(* IEC 61131-3 sources: verifaps-lib/share/xPPU (part 14) *)

        STEP White : (*Local Id: 11 *)
            Set_PriorityWhite(N);
        END_STEP

        STEP Conveyor : (*Local Id: 15 *)
        END_STEP

        STEP Black : (*Local Id: 26 *)
            Set_PriorityBlack(N);
        END_STEP

        STEP Ramp_End : (*Local Id: 30 *)
        END_STEP

        STEP Metallic : (*Local Id: 43 *)
            Set_PriorityMetallic(N);
        END_STEP

        STEP SetTargetChanged : (*Local Id: 53 *)
        END_STEP
        TRANSITION FROM (ResetTargets) TO (White) := (WPType_White); END_TRANSITION
        TRANSITION FROM (ResetTargets) TO (Black) := (WPType_Black); END_TRANSITION
        TRANSITION FROM (ResetTargets) TO (Metallic) := (WPType_Metallic); END_TRANSITION
        TRANSITION FROM (ResetTargets) TO (White) := (WPType_White); END_TRANSITION
        TRANSITION FROM (ResetTargets) TO (Black) := (WPType_Black); END_TRANSITION
        TRANSITION FROM (White) TO (Conveyor) := (Priority_White=1); END_TRANSITION
        TRANSITION FROM (White) TO (Ramp_End) := (Priority_White=2); END_TRANSITION
        TRANSITION FROM (Black) TO (Ramp_End) := (Priority_Black=2); END_TRANSITION
        TRANSITION FROM (Black) TO (Conveyor) := (Priority_Black=1); END_TRANSITION
        TRANSITION FROM (Metallic) TO (Conveyor) := (Priority_Metallic=1); END_TRANSITION
        TRANSITION FROM (Metallic) TO (Ramp_End) := (Priority_Metallic=2); END_TRANSITION
        TRANSITION FROM (Conveyor) TO (SetTargetChanged) := (CurrentTarget_Conveyor); END_TRANSITION
        TRANSITION FROM (Ramp_End) TO (SetTargetChanged) := (CurrentTarget_Conveyor); END_TRANSITION
        TRANSITION FROM (Ramp_End) TO (SetTargetChanged) := (CurrentTarget_Ramp); END_TRANSITION
        TRANSITION FROM (Conveyor) TO (SetTargetChanged) := (CurrentTarget_Ramp); END_TRANSITION
        TRANSITION FROM (Conveyor) TO (SetTargetChanged) := (CurrentTarget_Conveyor); END_TRANSITION
        TRANSITION FROM (Ramp_End) TO (SetTargetChanged) := (CurrentTarget_Conveyor); END_TRANSITION
        TRANSITION FROM (Conveyor) TO (SetTargetChanged) := (CurrentTarget_Conveyor); END_TRANSITION
        TRANSITION FROM (Ramp_End) TO (SetTargetChanged) := (CurrentTarget_Conveyor); END_TRANSITION
        TRANSITION FROM (ACT_ChangeTarget_Init) TO (ResetTargets) := (NOT TargetChanged AND NOT GVL.IsSFCResetting); END_TRANSITION
        TRANSITION FROM (SetTargetChanged) TO (ACT_ChangeTarget_Init) := (TargetChanged); END_TRANSITION
    END_ACTION
    ACTION ACT_CheckWPType

        INITIAL_STEP Conveyor_ACT_CheckWPType_Init : (*Local Id: 0 *)
        END_STEP

        STEP Reset_WPType : (*Local Id: 3 *)
        END_STEP

        STEP Wait_a_little_bit : (*Local Id: 11 *)
        END_STEP

        STEP WP_Is_White : (*Local Id: 15 *)
        END_STEP

        STEP WP_Is_Metallic : (*Local Id: 22 *)
        END_STEP

        STEP WP_Is_Black : (*Local Id: 30 *)
        END_STEP

        STEP WP_Type_Checked : (*Local Id: 36 *)
        END_STEP
        TRANSITION FROM (Reset_WPType) TO (Wait_a_little_bit) := (OptSensor.DI_WPLight); END_TRANSITION
        TRANSITION FROM (Reset_WPType) TO (WP_Is_Black) := (Reset_WPType.t>T#1s AND NOT IndSensor.DI_WPMetallic AND NOT OptSensor.DI_WPLight); END_TRANSITION
        TRANSITION FROM (Wait_a_little_bit) TO (WP_Is_White) := (Wait_a_little_bit.t>T#100ms AND NOT IndSensor.DI_WPMetallic); END_TRANSITION
        TRANSITION FROM (Wait_a_little_bit) TO (WP_Is_Metallic) := (IndSensor.DI_WPMetallic); END_TRANSITION
        TRANSITION FROM (WP_Is_White) TO (WP_Type_Checked) := (WPType_White); END_TRANSITION
        TRANSITION FROM (WP_Is_Metallic) TO (WP_Type_Checked) := (WPType_Metallic); END_TRANSITION
        TRANSITION FROM (WP_Is_White) TO (WP_Type_Checked) := (WPType_White); END_TRANSITION
        TRANSITION FROM (WP_Is_Metallic) TO (WP_Type_Checked) := (WPType_Metallic); END_TRANSITION
        TRANSITION FROM (WP_Is_Black) TO (WP_Type_Checked) := (WPType_Black); END_TRANSITION
        TRANSITION FROM (Conveyor_ACT_CheckWPType_Init) TO (Reset_WPType) := (NOT WPTypeChecked AND NOT GVL.IsSFCResetting); END_TRANSITION
        TRANSITION FROM (WP_Type_Checked) TO (Conveyor_ACT_CheckWPType_Init) := (WPTypeChecked); END_TRANSITION
    END_ACTION
    ACTION ACT_SortWP

        INITIAL_STEP Init_ACT_SortWP : (*Local Id: 0 *)
        END_STEP

        STEP ConveyorForwards : (*Local Id: 3 *)
            Motor.ACT_TurnClockwise(N);
        END_STEP

        STEP Wait : (*Local Id: 6 *)
        END_STEP

        STEP Checking_WP_Type : (*Local Id: 9 *)
            ACT_CheckWPType(N);
        END_STEP

        STEP Changing_Target : (*Local Id: 12 *)
            ACT_ChangeTarget(N);
        END_STEP

        STEP Chose_Right_Destination : (*Local Id: 15 *)
        END_STEP

        STEP Switch_Extending : (*Local Id: 19 *)
            Switch.ACT_Extend(N);
        END_STEP

        STEP Allow_FollowConveyorToOperate : (*Local Id: 22 *)
        END_STEP

        STEP Wait2sec : (*Local Id: 27 *)
        END_STEP

        STEP Stop_Allowence : (*Local Id: 30 *)
        END_STEP

        STEP Switch_Retracting : (*Local Id: 35 *)
            Switch.ACT_Retract(N);
        END_STEP

        STEP Transporting_To_Ramp : (*Local Id: 40 *)
        END_STEP

        STEP TurnConveyorOff : (*Local Id: 44 *)
            Motor.ACT_Stop(N);
        END_STEP

        STEP WP_Is_Sorted : (*Local Id: 47 *)
        END_STEP
        TRANSITION FROM (Chose_Right_Destination) TO (Switch_Extending) := (CurrentTarget_Conveyor); END_TRANSITION
        TRANSITION FROM (Chose_Right_Destination) TO (Transporting_To_Ramp) := (CurrentTarget_Ramp); END_TRANSITION
        TRANSITION FROM (Switch_Retracting) TO (TurnConveyorOff) := (Switch.Retracted); END_TRANSITION
        TRANSITION FROM (Transporting_To_Ramp) TO (TurnConveyorOff) := (Transporting_To_Ramp.t>T#2s); END_TRANSITION
        TRANSITION FROM (Init_ACT_SortWP) TO (ConveyorForwards) := (NOT WPSorted AND NOT GVL.IsSFCResetting); END_TRANSITION
        TRANSITION FROM (ConveyorForwards) TO (Wait) := (Motor.TurningClockwise); END_TRANSITION
        TRANSITION FROM (Wait) TO (Checking_WP_Type) := (Wait.t>T#900ms OR IndSensor.DI_WPMetallic OR OptSensor.DI_WPLight); END_TRANSITION
        TRANSITION FROM (Checking_WP_Type) TO (Changing_Target) := (WPTypeChecked); END_TRANSITION
        TRANSITION FROM (Changing_Target) TO (Chose_Right_Destination) := (TargetChanged); END_TRANSITION
        TRANSITION FROM (Switch_Extending) TO (Allow_FollowConveyorToOperate) := (Switch.Extended); END_TRANSITION
        TRANSITION FROM (Allow_FollowConveyorToOperate) TO (Wait2sec) := (FollowConveyor_AllowedToOperate); END_TRANSITION
        TRANSITION FROM (Wait2sec) TO (Stop_Allowence) := (Wait2sec.t>T#2s); END_TRANSITION
        TRANSITION FROM (Stop_Allowence) TO (Switch_Retracting) := (NOT FollowConveyor_AllowedToOperate); END_TRANSITION
        TRANSITION FROM (TurnConveyorOff) TO (WP_Is_Sorted) := (Motor.Stopped); END_TRANSITION
        TRANSITION FROM (WP_Is_Sorted) TO (Init_ACT_SortWP) := (WPSorted); END_TRANSITION
    END_ACTION
    ACTION ACT_AutomaticExecute

        INITIAL_STEP SmallSortingConveyor_ACT_AutomaticExecute_Init : (*Local Id: 0 *)
        END_STEP

        STEP Interstep : (*Local Id: 3 *)
        END_STEP

        STEP Sort_WP : (*Local Id: 11 *)
            ACT_SortWP(N);
        END_STEP

        STEP SetAutomaticExecuteCompleted : (*Local Id: 14 *)
        END_STEP
        TRANSITION FROM (Interstep) TO (Sort_WP) := (Check_AllowedToOperate AND Interstep.t>T#500ms); END_TRANSITION
        TRANSITION FROM (Interstep) TO (SmallSortingConveyor_ACT_AutomaticExecute_Init) := (NOT Check_AllowedToOperate AND Interstep.t>T#500ms); END_TRANSITION
        TRANSITION FROM (Interstep) TO (Sort_WP) := (Check_AllowedToOperate AND Interstep.t>T#500ms); END_TRANSITION
        TRANSITION FROM (SmallSortingConveyor_ACT_AutomaticExecute_Init) TO (Interstep) := (Check_AllowedToOperate AND NOT AutomaticExecuteCompleted AND NOT GVL.IsSFCResetting); END_TRANSITION
        TRANSITION FROM (Sort_WP) TO (SetAutomaticExecuteCompleted) := (WPSorted); END_TRANSITION
        TRANSITION FROM (SetAutomaticExecuteCompleted) TO (SmallSortingConveyor_ACT_AutomaticExecute_Init) := (AutomaticExecuteCompleted); END_TRANSITION
    END_ACTION
    ACTION ACT_EmergencyStop

        INITIAL_STEP Conveyor_ACT_EmergencyStop_Init : (*Local Id: 0 *)
        END_STEP

        STEP ResetVariables : (*Local Id: 3 *)
            Reset_Variables(N);
        END_STEP

        STEP Stop_Conveyor : (*Local Id: 6 *)
            Motor.ACT_Stop(N);
        END_STEP

        STEP Retract_Switch : (*Local Id: 9 *)
            Switch.ACT_Retract(N);
        END_STEP

        STEP Conveyor_EmergencyHandled : (*Local Id: 12 *)
        END_STEP
        TRANSITION FROM (Conveyor_ACT_EmergencyStop_Init) TO (ResetVariables) := (Not EmergencyHandled AND NOT GVL.IsSFCResetting); END_TRANSITION
        TRANSITION FROM (ResetVariables) TO (Stop_Conveyor) := (NOT InitCompleted AND NOT AutomaticExecuteCompleted); END_TRANSITION
        TRANSITION FROM (Stop_Conveyor) TO (Retract_Switch) := (Motor.Stopped); END_TRANSITION
        TRANSITION FROM (Retract_Switch) TO (Conveyor_EmergencyHandled) := (Switch.Retracted); END_TRANSITION
        TRANSITION FROM (Conveyor_EmergencyHandled) TO (Conveyor_ACT_EmergencyStop_Init) := (EmergencyHandled); END_TRANSITION
    END_ACTION
    ACTION ACT_Init

        INITIAL_STEP Init_ACT_Init : (*Local Id: 0 *)
        END_STEP

        STEP Interstep : (*Local Id: 5 *)
        END_STEP

        STEP ConveyorForwards : (*Local Id: 13 *)
            Motor.ACT_TurnClockwise(N);
        END_STEP

        STEP ExtendSwitch : (*Local Id: 16 *)
            Switch.ACT_Extend(N);
        END_STEP

        STEP Allow_FollowConveyorToInit : (*Local Id: 19 *)
            Set_FollowConveyorAllowedToInit(P0);
            Reset_FollowConveyorAllowedToInit(P1);
        END_STEP

        STEP RetractSwitch : (*Local Id: 22 *)
            Switch.ACT_Retract(N);
        END_STEP

        STEP Stop_Conveyors : (*Local Id: 25 *)
            Motor.ACT_Stop(N);
        END_STEP

        STEP SetInitCompleted : (*Local Id: 28 *)
        END_STEP
        TRANSITION FROM (Interstep) TO (ConveyorForwards) := (Check_AllowedToInit AND NOT InitCompleted AND Interstep.t>T#500ms); END_TRANSITION
        TRANSITION FROM (Interstep) TO (Init_ACT_Init) := ((NOT Check_AllowedToInit OR InitCompleted) AND Interstep.t>T#500ms); END_TRANSITION
        TRANSITION FROM (Interstep) TO (ConveyorForwards) := (Check_AllowedToInit AND NOT InitCompleted AND Interstep.t>T#500ms); END_TRANSITION
        TRANSITION FROM (Init_ACT_Init) TO (Interstep) := (Check_AllowedToInit AND NOT InitCompleted AND NOT GVL.IsSFCResetting); END_TRANSITION
        TRANSITION FROM (ConveyorForwards) TO (ExtendSwitch) := (Motor.TurningClockwise); END_TRANSITION
        TRANSITION FROM (ExtendSwitch) TO (Allow_FollowConveyorToInit) := (Switch.Extended); END_TRANSITION
        TRANSITION FROM (Allow_FollowConveyorToInit) TO (RetractSwitch) := (Check_FollowConveyor_InitCompleted); END_TRANSITION
        TRANSITION FROM (RetractSwitch) TO (Stop_Conveyors) := (Switch.Retracted); END_TRANSITION
        TRANSITION FROM (Stop_Conveyors) TO (SetInitCompleted) := (Motor.Stopped); END_TRANSITION
        TRANSITION FROM (SetInitCompleted) TO (Init_ACT_Init) := (InitCompleted); END_TRANSITION
    END_ACTION

    Check_AllowedToInit := Main.Check_SmallSortingConveyor_AllowedToInit;
    Check_AllowedToOperate := Main.Check_SmallSortingConveyor_AllowedToOperate;
    Check_FollowConveyor_InitCompleted := Main.Check_SmallSortingConveyor_FollowConveyor_InitCompleted;
    Check_FollowConveyor_AutomaticExecuteCompleted := Main.Check_SmallSortingConveyor_FollowConveyor_AutomaticExecuteCompleted;
END_FUNCTION_BLOCK

FUNCTION_BLOCK Stack

    VAR_INPUT
        Seperator : MonostableCylinder;
        Panel : OperationPanel;
        WPAvailable : MicroSwitch;
        InductiveSensor : InductiveSensor;
        OpticalSensor : OpticalSensor;
        WeightModule : WeightModule;
        Check_WPPickedUp : BOOL;
        SFCReset : BOOL;
    END_VAR

    VAR_OUTPUT
        StartButton : BOOL;
        InitCompleted : BOOL;
        AutomaticExecuteCompleted : BOOL;
        EmergencyStop : BOOL;
        EmergencyHandled : BOOL;
    END_VAR

    VAR
        WPProvided : BOOL;
        WPType_White : BOOL;
        WPType_Black : BOOL;
        WPType_Metallic : BOOL;
        WPWeight_Light : BOOL;
        WPWeight_Medium : BOOL;
        WPWeight_Heavy : BOOL;
        Timer : TON;
        SFCInit : BOOL;
    END_VAR
    ACTION Reset_Timer

        Timer(IN:=FALSE);
    END_ACTION
    ACTION Reset_Variables

        InitCompleted := FALSE;
        AutomaticExecuteCompleted := FALSE;

        WPType_White:=FALSE;
        WPType_Black:=FALSE;
        WPType_Metallic:=FALSE;
        WPWeight_Light:=FALSE;
        WPWeight_Medium:=FALSE;
        WPWeight_Heavy:=FALSE;
    END_ACTION
    ACTION Set_Timer250ms

        Timer(IN:=TRUE, PT:=T#250MS);
    END_ACTION
    ACTION Set_WPParameters_AND_WPProvided

        //WPType
        IF(NOT InductiveSensor.DI_WPMetallic AND NOT OpticalSensor.DI_WPLight)THEN
        	WPType_Black:=TRUE;
        	WPType_White:=FALSE;
        	WPType_Metallic:=FALSE;
        ELSIF(NOT InductiveSensor.DI_WPMetallic AND OpticalSensor.DI_WPLight)THEN
        	WPType_Black:=FALSE;
        	WPType_White:=TRUE;
        	WPType_Metallic:=FALSE;
        ELSIF(InductiveSensor.DI_WPMetallic)THEN
        	WPType_Black:=FALSE;
        	WPType_White:=FALSE;
        	WPType_Metallic:=TRUE;
        END_IF
        //WPWeight
        IF(WeightModule.AI_WPWeight<12000)THEN
        	WPWeight_Light:=TRUE;
        	WPWeight_Medium:=FALSE;
        	WPWeight_Heavy:=FALSE;
        ELSIF(12000<=WeightModule.AI_WPWeight AND WeightModule.AI_WPWeight<24000)THEN
        	WPWeight_Light:=FALSE;
        	WPWeight_Medium:=TRUE;
        	WPWeight_Heavy:=FALSE;
        ELSIF(2400<=WeightModule.AI_WPWeight)THEN
        	WPWeight_Light:=FALSE;
        	WPWeight_Medium:=FALSE;
        	WPWeight_Heavy:=TRUE;
        END_IF

        WPProvided:=TRUE;
    END_ACTION
    ACTION ACT_ProvideWP

        INITIAL_STEP ACT_ProvideWP_Init : (*Local Id: 0 *)
        END_STEP

        STEP Slider_Extend : (*Local Id: 3 *)
            Seperator.ACT_Extend(N);
        END_STEP

        STEP WP_Ready : (*Local Id: 6 *)
        END_STEP

        STEP Black : (*Local Id: 17 *)
        END_STEP

        STEP Light : (*Local Id: 22 *)
        END_STEP

        STEP White : (*Local Id: 29 *)
        END_STEP

        STEP Metallic : (*Local Id: 37 *)
        END_STEP

        STEP Weight_Choice : (*Local Id: 42 *)
        END_STEP

        STEP Medium : (*Local Id: 49 *)
        END_STEP

        STEP Heavy : (*Local Id: 56 *)
        END_STEP

        STEP WP_Provided : (*Local Id: 63 *)
        END_STEP
        TRANSITION FROM (WP_Ready) TO (Black) := (NOT InductiveSensor.DI_WPMetallic AND NOT OpticalSensor.DI_WPLight); END_TRANSITION
        TRANSITION FROM (WP_Ready) TO (White) := (NOT InductiveSensor.DI_WPMetallic AND OpticalSensor.DI_WPLight); END_TRANSITION
        TRANSITION FROM (WP_Ready) TO (Metallic) := (InductiveSensor.DI_WPMetallic); END_TRANSITION
        TRANSITION FROM (Weight_Choice) TO (Light) := (WeightModule.AI_WPWeight<12000); END_TRANSITION
        TRANSITION FROM (Weight_Choice) TO (Medium) := (12000<=WeightModule.AI_WPWeight AND WeightModule.AI_WPWeight<24000); END_TRANSITION
        TRANSITION FROM (Weight_Choice) TO (Heavy) := (2400<=WeightModule.AI_WPWeight); END_TRANSITION
        TRANSITION FROM (Medium) TO (WP_Provided) := (WPWeight_Medium); END_TRANSITION
        TRANSITION FROM (Heavy) TO (WP_Provided) := (WPWeight_Heavy); END_TRANSITION
        TRANSITION FROM (Light) TO (WP_Provided) := (WPWeight_Light); END_TRANSITION
        TRANSITION FROM (Medium) TO (WP_Provided) := (WPWeight_Medium); END_TRANSITION
        TRANSITION FROM (Heavy) TO (WP_Provided) := (WPWeight_Heavy); END_TRANSITION
        TRANSITION FROM (ACT_ProvideWP_Init) TO (Slider_Extend) := (NOT WPAvailable.DI_SwitchTrue AND NOT GVL.IsSFCResetting); END_TRANSITION
        TRANSITION FROM (Slider_Extend) TO (WP_Ready) := (Seperator.Extended AND WPAvailable.DI_SwitchTrue); END_TRANSITION
        TRANSITION FROM (Black) TO (Light) := (WPType_Black); END_TRANSITION
        TRANSITION FROM (White) TO (Light) := (WPType_White); END_TRANSITION
        TRANSITION FROM (Metallic) TO (Weight_Choice) := (WPType_Metallic); END_TRANSITION
        TRANSITION FROM (WP_Provided) TO (ACT_ProvideWP_Init) := (WPProvided); END_TRANSITION
    END_ACTION
    ACTION ACT_AutomaticExecute

        INITIAL_STEP ACT_AutomaticExecute_Init : (*Local Id: 0 *)
        END_STEP

        STEP Short_Delay : (*Local Id: 3 *)
            Reset_Timer(P0);
            Set_Timer250ms(N);
        END_STEP

        STEP Provide_WP : (*Local Id: 7 *)
            ACT_ProvideWP(N);
        END_STEP

        STEP Dont_Provide_WP : (*Local Id: 12 *)
        END_STEP

        STEP Waiting_For_Crane_To_Pick_Up : (*Local Id: 18 *)
        END_STEP

        STEP Stack_Retracing : (*Local Id: 21 *)
            Seperator.ACT_Retract(N);
        END_STEP
        TRANSITION FROM (Short_Delay) TO (Provide_WP) := (Timer.Q AND NOT WPAvailable.DI_SwitchTrue); END_TRANSITION
        TRANSITION FROM (Short_Delay) TO (Dont_Provide_WP) := (Timer.Q AND WPAvailable.DI_SwitchTrue); END_TRANSITION
        TRANSITION FROM (Provide_WP) TO (Waiting_For_Crane_To_Pick_Up) := (WPProvided); END_TRANSITION
        TRANSITION FROM (Dont_Provide_WP) TO (Waiting_For_Crane_To_Pick_Up) := (WPProvided); END_TRANSITION
        TRANSITION FROM (ACT_AutomaticExecute_Init) TO (Short_Delay) := (NOT AutomaticExecuteCompleted AND NOT GVL.IsSFCResetting); END_TRANSITION
        TRANSITION FROM (Waiting_For_Crane_To_Pick_Up) TO (Stack_Retracing) := (NOT WPAvailable.DI_SwitchTrue AND Check_WPPickedUp); END_TRANSITION
        TRANSITION FROM (Stack_Retracing) TO (ACT_AutomaticExecute_Init) := (Seperator.Retracted); END_TRANSITION
    END_ACTION
    ACTION ACT_EmergencyStop

        INITIAL_STEP Magazine_ACT_EmergencyStop_Init : (*Local Id: 0 *)
        END_STEP

        STEP ResetVariables : (*Local Id: 3 *)
            Reset_Variables(N);
        END_STEP

        STEP Stack_Retracting : (*Local Id: 6 *)
            Seperator.ACT_Retract(N);
        END_STEP

        STEP Stack_EmergencyHandled : (*Local Id: 9 *)
        END_STEP
        TRANSITION FROM (Magazine_ACT_EmergencyStop_Init) TO (ResetVariables) := (Not EmergencyHandled AND NOT GVL.IsSFCResetting); END_TRANSITION
        TRANSITION FROM (ResetVariables) TO (Stack_Retracting) := (NOT InitCompleted AND NOT AutomaticExecuteCompleted); END_TRANSITION
        TRANSITION FROM (Stack_Retracting) TO (Stack_EmergencyHandled) := (Seperator.Retracted); END_TRANSITION
        TRANSITION FROM (Stack_EmergencyHandled) TO (Magazine_ACT_EmergencyStop_Init) := (EmergencyHandled); END_TRANSITION
    END_ACTION
    ACTION ACT_Init

        INITIAL_STEP Stack_ACT_Init : (*Local Id: 0 *)
        END_STEP

        STEP Set_WP_Parameters : (*Local Id: 6 *)
            Set_WPParameters_AND_WPProvided(N);
        END_STEP

        STEP Retract_Cylinder_Init : (*Local Id: 10 *)
            Seperator.ACT_Retract(N);
        END_STEP

        STEP SetInitCompleted : (*Local Id: 13 *)
        END_STEP
        TRANSITION FROM (Stack_ACT_Init) TO (Retract_Cylinder_Init) := (NOT InitCompleted AND NOT WPAvailable.DI_SwitchTrue AND NOT GVL.IsSFCResetting); END_TRANSITION
        TRANSITION FROM (Stack_ACT_Init) TO (Set_WP_Parameters) := (NOT InitCompleted AND WPAvailable.DI_SwitchTrue AND NOT GVL.IsSFCResetting); END_TRANSITION
        TRANSITION FROM (Stack_ACT_Init) TO (Retract_Cylinder_Init) := (NOT InitCompleted AND NOT WPAvailable.DI_SwitchTrue AND NOT GVL.IsSFCResetting); END_TRANSITION
        TRANSITION FROM (Set_WP_Parameters) TO (Retract_Cylinder_Init) := (WPProvided); END_TRANSITION
        TRANSITION FROM (Retract_Cylinder_Init) TO (SetInitCompleted) := (Seperator.Retracted); END_TRANSITION
        TRANSITION FROM (SetInitCompleted) TO (Stack_ACT_Init) := (InitCompleted); END_TRANSITION
    END_ACTION

    Panel();
    StartButton := Panel.StartButton;
    EmergencyStop := Panel.EmergencyStop;
    Check_WPPickedUp := Main.Check_Stack_WPPickedUp;
END_FUNCTION_BLOCK

FUNCTION_BLOCK Stamp

    VAR_INPUT
        Panel : OperationPanel;
        PressureSensor : PressureSensor;
        PropValve : ProportionalValve;
        WPAvailable : MicroSwitch;
        StampingCylinder : MonostableCylinder;
        SlidingCylinder : BistableCylinder;
        SoftwareEmergency : BOOL;
        Check_Allowed_To_Operate : BOOL;
        Check_WPWeight_Light : BOOL;
        Check_WPWeight_Medium : BOOL;
        Check_WPWeight_Heavy : BOOL;
        SFCReset : BOOL;
    END_VAR

    VAR_OUTPUT
        StartButton : BOOL;
        InitCompleted : BOOL;
        AutomaticExecuteCompleted : BOOL;
        EmergencyStop : BOOL;
        EmergencyHandled : BOOL;
        IsStamping : BOOL;
    END_VAR

    VAR
        WPStamped : BOOL;
        WPType_White : BOOL;
        WPType_Black : BOOL;
        WPType_Metallic : BOOL;
        WPWeight_Light : BOOL;
        WPWeight_Medium : BOOL;
        WPWeight_Heavy : BOOL;
        Timer : TON;
        SFCInit : BOOL;
    END_VAR
    ACTION ExtendStampingCylinder_AND_Timer1500ms

        StampingCylinder.ACT_Extend();
        Timer(IN:=TRUE, PT:=T#1500MS);
    END_ACTION
    ACTION Reset_Pressure

        PropValve.AO_SetPressure:=0;
    END_ACTION
    ACTION Reset_Timer

        Timer(IN:=FALSE);
    END_ACTION
    ACTION Reset_Variables

        InitCompleted := FALSE;
        AutomaticExecuteCompleted := FALSE;

        propValve.AO_SetPressure:=0;
        IsStamping:=FALSE;
        WPStamped:=FALSE;
        WPType_Black := FALSE;
        WPType_White := FALSE;
        WPType_Metallic := FALSE;
        WPWeight_Light := FALSE;
        WPWeight_Medium := FALSE;
        WPWeight_Heavy := FALSE;
    END_ACTION
    ACTION Set_HeavyPressure

        PropValve.AO_SetPressure:=7000;
    END_ACTION
    ACTION Set_LightPressure

        PropValve.AO_SetPressure:=4000;
    END_ACTION
    ACTION Set_MediumPressure

        PropValve.AO_SetPressure:=5500;
    END_ACTION
    ACTION Set_Timer1000ms

        Timer(IN:=TRUE, PT:=T#1000MS);
    END_ACTION
    ACTION Set_Timer500ms

        Timer(IN:=TRUE, PT:=T#500ms);
    END_ACTION
    ACTION Set_WPWeight

        WPWeight_Light := Check_WPWeight_Light;
        WPWeight_Medium := Check_WPWeight_Medium;
        WPWeight_Heavy := Check_WPWeight_Heavy;
    END_ACTION
    ACTION ACT_Stamp

        INITIAL_STEP Stamp_ACT_Stamp : (*Local Id: 0 *)
        END_STEP

        STEP Get_WPWeight_From_Crane : (*Local Id: 3 *)
            Set_WPWeight(N);
        END_STEP

        STEP Slider_Retract : (*Local Id: 6 *)
            SlidingCylinder.ACT_Retract(N);
        END_STEP

        STEP SetLightPressure : (*Local Id: 10 *)
            Set_LightPressure(N);
        END_STEP

        STEP SetMediumPressure : (*Local Id: 15 *)
            Set_MediumPressure(N);
        END_STEP

        STEP SetHeavyPressure : (*Local Id: 20 *)
            Set_HeavyPressure(N);
        END_STEP

        STEP Extend_StampingCylinder : (*Local Id: 24 *)
            Reset_Timer(P0);
            ExtendStampingCylinder_AND_Timer1500ms(N);
        END_STEP

        STEP CheckCorrectPressure : (*Local Id: 28 *)
        END_STEP

        STEP HeavyPressureOk : (*Local Id: 32 *)
        END_STEP

        STEP MediumPressureOk : (*Local Id: 37 *)
        END_STEP

        STEP LightPressureOk : (*Local Id: 42 *)
        END_STEP

        STEP Error : (*Local Id: 48 *)
        END_STEP

        STEP Wait : (*Local Id: 55 *)
            Reset_Timer(P0);
            Set_Timer1000ms(N);
        END_STEP

        STEP ResetPressure : (*Local Id: 58 *)
            Reset_Pressure(N);
        END_STEP

        STEP Move_Stamp_Up : (*Local Id: 61 *)
            StampingCylinder.ACT_Retract(N);
        END_STEP

        STEP Slider_Extend : (*Local Id: 64 *)
            SlidingCylinder.ACT_Extend(N);
        END_STEP

        STEP WP_Stamped : (*Local Id: 67 *)
        END_STEP
        TRANSITION FROM (Slider_Retract) TO (SetLightPressure) := (SlidingCylinder.Retracted AND WPWeight_Light); END_TRANSITION
        TRANSITION FROM (Slider_Retract) TO (SetMediumPressure) := (SlidingCylinder.Retracted AND WPWeight_Medium); END_TRANSITION
        TRANSITION FROM (Slider_Retract) TO (SetHeavyPressure) := (SlidingCylinder.Retracted AND WPWeight_Heavy); END_TRANSITION
        TRANSITION FROM (Extend_StampingCylinder) TO (CheckCorrectPressure) := (StampingCylinder.Extended); END_TRANSITION
        TRANSITION FROM (Extend_StampingCylinder) TO (Error) := (Timer.Q); END_TRANSITION
        TRANSITION FROM (CheckCorrectPressure) TO (HeavyPressureOk) := ((PressureSensor.AI_CurrentPressure > 18000) AND WPWeight_Heavy); END_TRANSITION
        TRANSITION FROM (CheckCorrectPressure) TO (MediumPressureOk) := ((PressureSensor.AI_CurrentPressure > 5300) AND (PressureSensor.AI_CurrentPressure < 17000) AND WPWeight_Medium); END_TRANSITION
        TRANSITION FROM (CheckCorrectPressure) TO (LightPressureOk) := ((PressureSensor.AI_CurrentPressure > 4800) AND (PressureSensor.AI_CurrentPressure < 5200) AND WPWeight_Light); END_TRANSITION
        TRANSITION FROM (SetLightPressure) TO (Extend_StampingCylinder) := (PropValve.AO_SetPressure=4000); END_TRANSITION
        TRANSITION FROM (SetMediumPressure) TO (Extend_StampingCylinder) := (PropValve.AO_SetPressure=5500); END_TRANSITION
        TRANSITION FROM (SetHeavyPressure) TO (Extend_StampingCylinder) := (PropValve.AO_SetPressure=7000); END_TRANSITION
        TRANSITION FROM (HeavyPressureOk) TO (Wait) := (TRUE); END_TRANSITION
        TRANSITION FROM (MediumPressureOk) TO (Wait) := (TRUE); END_TRANSITION
        TRANSITION FROM (LightPressureOk) TO (Wait) := (TRUE); END_TRANSITION
        TRANSITION FROM (HeavyPressureOk) TO (Wait) := (TRUE); END_TRANSITION
        TRANSITION FROM (MediumPressureOk) TO (Wait) := (TRUE); END_TRANSITION
        TRANSITION FROM (LightPressureOk) TO (Wait) := (TRUE); END_TRANSITION
        TRANSITION FROM (Stamp_ACT_Stamp) TO (Get_WPWeight_From_Crane) := (IsStamping AND NOT WPStamped AND WPAvailable.DI_SwitchTrue AND NOT GVL.IsSFCResetting); END_TRANSITION
        TRANSITION FROM (Get_WPWeight_From_Crane) TO (Slider_Retract) := (WPWeight_Light=Check_WPWeight_Light AND WPWeight_Medium=Check_WPWeight_Medium AND WPWeight_Heavy=Check_WPWeight_Heavy); END_TRANSITION
        TRANSITION FROM (Error) TO (Stamp_ACT_Stamp) := (SoftwareEmergency); END_TRANSITION
        TRANSITION FROM (Wait) TO (ResetPressure) := (Timer.Q); END_TRANSITION
        TRANSITION FROM (ResetPressure) TO (Move_Stamp_Up) := (PropValve.AO_SetPressure=0); END_TRANSITION
        TRANSITION FROM (Move_Stamp_Up) TO (Slider_Extend) := (StampingCylinder.Retracted); END_TRANSITION
        TRANSITION FROM (Slider_Extend) TO (WP_Stamped) := (SlidingCylinder.Extended); END_TRANSITION
        TRANSITION FROM (WP_Stamped) TO (Stamp_ACT_Stamp) := (WPStamped); END_TRANSITION
    END_ACTION
    ACTION ACT_AutomaticExecute

        INITIAL_STEP Stamp_AutomaticExecute_Init : (*Local Id: 0 *)
        END_STEP

        STEP Dummy1 : (*Local Id: 3 *)
        END_STEP

        STEP Dummy2 : (*Local Id: 6 *)
        END_STEP

        STEP Intersetp : (*Local Id: 9 *)
            Reset_Timer(P0);
            Set_Timer500ms(N);
        END_STEP

        STEP PrepareStamping : (*Local Id: 12 *)
        END_STEP

        STEP Stamp_WP : (*Local Id: 18 *)
            ACT_Stamp(N);
        END_STEP

        STEP SetAutomaticExecuteCompleted : (*Local Id: 21 *)
        END_STEP
        TRANSITION FROM (Stamp_AutomaticExecute_Init) TO (Dummy1) := (NOT AutomaticExecuteCompleted AND NOT GVL.IsSFCResetting); END_TRANSITION
        TRANSITION FROM (Dummy1) TO (Dummy2) := (NOT WPAvailable.DI_SwitchTrue); END_TRANSITION
        TRANSITION FROM (Dummy2) TO (Intersetp) := (Check_Allowed_To_Operate AND WPAvailable.DI_SwitchTrue); END_TRANSITION
        TRANSITION FROM (Intersetp) TO (PrepareStamping) := (Check_Allowed_To_Operate AND Timer.Q); END_TRANSITION
        TRANSITION FROM (PrepareStamping) TO (Stamp_WP) := (IsStamping AND NOT WPStamped); END_TRANSITION
        TRANSITION FROM (Stamp_WP) TO (SetAutomaticExecuteCompleted) := (WPStamped); END_TRANSITION
        TRANSITION FROM (SetAutomaticExecuteCompleted) TO (Stamp_AutomaticExecute_Init) := (AutomaticExecuteCompleted); END_TRANSITION
    END_ACTION
    ACTION ACT_EmergencyStop

        INITIAL_STEP Stamp_ACT_EmergencyStop_Init : (*Local Id: 0 *)
        END_STEP

        STEP ResetVariables : (*Local Id: 3 *)
            Reset_Variables(N);
        END_STEP

        STEP Stamp_Retracting : (*Local Id: 6 *)
            StampingCylinder.ACT_Retract(N);
        END_STEP

        STEP SlidingCylinder_Retracting : (*Local Id: 9 *)
            SlidingCylinder.ACT_Extend(N);
        END_STEP

        STEP Stamp_EmergencyHandled : (*Local Id: 12 *)
        END_STEP
        TRANSITION FROM (Stamp_ACT_EmergencyStop_Init) TO (ResetVariables) := (Not EmergencyHandled AND NOT GVL.IsSFCResetting); END_TRANSITION
        TRANSITION FROM (ResetVariables) TO (Stamp_Retracting) := (NOT InitCompleted AND NOT AutomaticExecuteCompleted); END_TRANSITION
        TRANSITION FROM (Stamp_Retracting) TO (SlidingCylinder_Retracting) := (StampingCylinder.Retracted); END_TRANSITION
        TRANSITION FROM (SlidingCylinder_Retracting) TO (Stamp_EmergencyHandled) := (SlidingCylinder.Extended); END_TRANSITION
        TRANSITION FROM (Stamp_EmergencyHandled) TO (Stamp_ACT_EmergencyStop_Init) := (EmergencyHandled); END_TRANSITION
    END_ACTION
    ACTION ACT_Init

        INITIAL_STEP Stamp_ACT_Init : (*Local Id: 0 *)
        END_STEP

        STEP Retract_Stamping_Cylinder_Init : (*Local Id: 3 *)
            StampingCylinder.ACT_Retract(N);
        END_STEP

        STEP Extend_Sliding_Cylinder_Init : (*Local Id: 6 *)
            SlidingCylinder.ACT_Extend(N);
        END_STEP

        STEP SetInitCompleted : (*Local Id: 9 *)
        END_STEP
        TRANSITION FROM (Stamp_ACT_Init) TO (Retract_Stamping_Cylinder_Init) := (NOT InitCompleted AND NOT GVL.IsSFCResetting); END_TRANSITION
        TRANSITION FROM (Retract_Stamping_Cylinder_Init) TO (Extend_Sliding_Cylinder_Init) := (StampingCylinder.Retracted); END_TRANSITION
        TRANSITION FROM (Extend_Sliding_Cylinder_Init) TO (SetInitCompleted) := (SlidingCylinder.Extended); END_TRANSITION
        TRANSITION FROM (SetInitCompleted) TO (Stamp_ACT_Init) := (InitCompleted); END_TRANSITION
    END_ACTION

    Panel();
    StartButton := Panel.StartButton;
    EmergencyStop := Panel.EmergencyStop;
    Check_Allowed_To_Operate := Main.Check_Stamp_AllowedToOperate;
    Check_WPWeight_Light:=Main.Crane_WPWeight_Light;
    Check_WPWeight_Medium:=Main.Crane_WPWeight_Medium;
    Check_WPWeight_Heavy:=Main.Crane_WPWeight_Heavy;
END_FUNCTION_BLOCK

FUNCTION_BLOCK Switch

    VAR_OUTPUT
        Extended : BOOL;
        Retracted : BOOL;
    END_VAR

    VAR
        DI_Extended : BOOL;
        DI_Retracted : BOOL;
        DO_Extend : BOOL;
        SFCInit : BOOL;
        SFCReset : BOOL;
    END_VAR
    ACTION ACT_Extend

        INITIAL_STEP Init_ACT_Extend : (*Local Id: 0 *)
        END_STEP

        STEP Extend_Cylinder : (*Local Id: 3 *)
        END_STEP

        STEP SetExtended : (*Local Id: 8 *)
        END_STEP
        TRANSITION FROM (Init_ACT_Extend) TO (Extend_Cylinder) := (NOT Extended AND NOT GVL.IsSFCResetting); END_TRANSITION
        TRANSITION FROM (Extend_Cylinder) TO (SetExtended) := (DI_Extended); END_TRANSITION
        TRANSITION FROM (SetExtended) TO (Init_ACT_Extend) := (Extended); END_TRANSITION
    END_ACTION
    ACTION ACT_Retract

        INITIAL_STEP Init_ACT_Retract : (*Local Id: 0 *)
        END_STEP

        STEP Retract_Cylinder : (*Local Id: 3 *)
        END_STEP

        STEP SetRetacted : (*Local Id: 8 *)
        END_STEP
        TRANSITION FROM (Init_ACT_Retract) TO (Retract_Cylinder) := (NOT Retracted AND NOT GVL.IsSFCResetting); END_TRANSITION
        TRANSITION FROM (Retract_Cylinder) TO (SetRetacted) := (DI_Retracted); END_TRANSITION
        TRANSITION FROM (SetRetacted) TO (Init_ACT_Retract) := (Retracted); END_TRANSITION
    END_ACTION

END_FUNCTION_BLOCK

FUNCTION_BLOCK TurningTable

    VAR
        Motor : Motor;
        AtStack : MicroSwitch;
        AtConveyor : MicroSwitch;
        AtStamp : MicroSwitch;
    END_VAR

END_FUNCTION_BLOCK

FUNCTION_BLOCK UltrasonicSensor

    VAR
        AI_UltraSonic : INT;
    END_VAR

END_FUNCTION_BLOCK

FUNCTION_BLOCK VacuumGripper

    VAR_INPUT
        Valve : Valve;
        VacuumSwitch : VacuumSwitch;
    END_VAR

    VAR_OUTPUT
        Intaken : BOOL;
        Released : BOOL;
    END_VAR

    VAR
        SFCInit : BOOL;
        SFCReset : BOOL;
    END_VAR
    ACTION ACT_Intake

        INITIAL_STEP Init_ACT_Intake : (*Local Id: 0 *)
        END_STEP

        STEP TurnVacuumOn : (*Local Id: 3 *)
            Valve.ACT_TurnVacuumOn(N);
        END_STEP

        STEP SetWPTakenIn : (*Local Id: 6 *)
        END_STEP
        TRANSITION FROM (Init_ACT_Intake) TO (TurnVacuumOn) := (NOT Intaken AND NOT GVL.IsSFCResetting); END_TRANSITION
        TRANSITION FROM (TurnVacuumOn) TO (SetWPTakenIn) := (VacuumSwitch.DI_TakenIn); END_TRANSITION
        TRANSITION FROM (SetWPTakenIn) TO (Init_ACT_Intake) := (Intaken); END_TRANSITION
    END_ACTION
    ACTION ACT_Release

        INITIAL_STEP Init_ACT_Release : (*Local Id: 0 *)
        END_STEP

        STEP TurnVacuumOff : (*Local Id: 3 *)
            Valve.ACT_TurnVacuumOff(N);
        END_STEP

        STEP SetWPReleased : (*Local Id: 6 *)
        END_STEP
        TRANSITION FROM (Init_ACT_Release) TO (TurnVacuumOff) := (NOT Released AND NOT GVL.IsSFCResetting); END_TRANSITION
        TRANSITION FROM (TurnVacuumOff) TO (SetWPReleased) := (NOT VacuumSwitch.DI_TakenIn); END_TRANSITION
        TRANSITION FROM (SetWPReleased) TO (Init_ACT_Release) := (Released); END_TRANSITION
    END_ACTION

END_FUNCTION_BLOCK

FUNCTION_BLOCK VacuumGripperExtended

    VAR_INPUT
        Valve : Valve;
        VacuumSwitch : VacuumSwitch;
    END_VAR

    VAR_OUTPUT
        Intaken : BOOL;
        Released : BOOL;
    END_VAR

    VAR
        DO_VacuumHit : BOOL;
        SFCInit : BOOL;
        SFCReset : BOOL;
    END_VAR
    ACTION ACT_Intake

        INITIAL_STEP Init_ACT_Intake : (*Local Id: 0 *)
        END_STEP

        STEP TurnVacuumOn : (*Local Id: 3 *)
            Valve.ACT_TurnVacuumOn(N);
        END_STEP

        STEP SetWPTakenIn : (*Local Id: 6 *)
        END_STEP
        TRANSITION FROM (Init_ACT_Intake) TO (TurnVacuumOn) := (NOT Intaken AND NOT GVL.IsSFCResetting); END_TRANSITION
        TRANSITION FROM (TurnVacuumOn) TO (SetWPTakenIn) := (VacuumSwitch.DI_TakenIn); END_TRANSITION
        TRANSITION FROM (SetWPTakenIn) TO (Init_ACT_Intake) := (Intaken); END_TRANSITION
    END_ACTION
    ACTION ACT_Release

        INITIAL_STEP Init_ACT_Release : (*Local Id: 0 *)
        END_STEP

        STEP TurnVacuumOff : (*Local Id: 3 *)
            Valve.ACT_TurnVacuumOff(N);
        END_STEP

        STEP SetWPReleased : (*Local Id: 8 *)
        END_STEP
        TRANSITION FROM (Init_ACT_Release) TO (TurnVacuumOff) := (NOT Released AND NOT GVL.IsSFCResetting); END_TRANSITION
        TRANSITION FROM (TurnVacuumOff) TO (SetWPReleased) := (NOT VacuumSwitch.DI_TakenIn AND TurnVacuumOff.t>T#250ms); END_TRANSITION
        TRANSITION FROM (SetWPReleased) TO (Init_ACT_Release) := (Released); END_TRANSITION
    END_ACTION

END_FUNCTION_BLOCK

FUNCTION_BLOCK VacuumSwitch

    VAR
        DI_TakenIn : BOOL;
    END_VAR

END_FUNCTION_BLOCK

FUNCTION_BLOCK Valve

    VAR
        DO_VacuumOn : BOOL;
    END_VAR
    ACTION ACT_TurnVacuumOff

        DO_VacuumOn := FALSE;
    END_ACTION
    ACTION ACT_TurnVacuumOn

        DO_VacuumOn := TRUE;
    END_ACTION

END_FUNCTION_BLOCK

FUNCTION_BLOCK WeightModule

    VAR
        AI_WPWeight : INT;
    END_VAR

END_FUNCTION_BLOCK

FUNCTION_BLOCK xPPU

    VAR_INPUT
        Stack : Stack;
        Crane : Crane;
        LargeSortingConveyor : LargeSortingConveyor;
        Stamp : Stamp;
        PicAlphaConveyor : PicAlphaConveyor;
        SmallSortingConveyor : SmallSortingConveyor;
        RefillConveyor : RefillConveyor;
        PicAlpha : PicAlpha;
        SafetyDoor : SafetyDoor;
        LightGrid : LightGrid;
        SFCReset : BOOL;
    END_VAR

    VAR_OUTPUT
        StartButton : BOOL;
        InitCompleted : BOOL;
        AutomaticExecuteCompleted : BOOL;
        EmergencyStop : BOOL;
        EmergencyHandled : BOOL;
        SFCResetResetCompleted : BOOL;
        SFCResetCompleted : BOOL;
    END_VAR

    VAR
        SFCInit : BOOL;
    END_VAR
    ACTION ACT_CheckEmergency

        EmergencyStop := Stack.EmergencyStop OR LargeSortingConveyor.EmergencyStop OR Stamp.EmergencyStop OR SafetyDoor.EmergencyStop OR LightGrid.EmergencyStop OR Crane.SoftwareEmergency OR Stamp.SoftwareEmergency OR PicAlpha.SoftwareEmergency;
    END_ACTION
    ACTION ACT_Start

        StartButton := Stack.StartButton OR LargeSortingConveyor.StartButton OR Stamp.StartButton OR SafetyDoor.StartButton OR LightGrid.StartButton;
    END_ACTION
    ACTION AutomaticExecute_entry

        AutomaticExecuteCompleted:=FALSE;

        LargeSortingConveyor.Panel.ACT_TurnLampWhite_Off();
        Stack.Panel.ACT_TurnLampWhite_Off();
        Stamp.Panel.ACT_TurnLampWhite_Off();
        LargeSortingConveyor.Panel.ACT_TurnLampGreen_On();
        Stack.Panel.ACT_TurnLampGreen_On();
        Stamp.Panel.ACT_TurnLampGreen_On();
    END_ACTION
    ACTION CallAll_AutomationExecutes

        EmergencyStop := Stack.EmergencyStop OR LargeSortingConveyor.EmergencyStop OR Stamp.EmergencyStop OR SafetyDoor.EmergencyStop OR LightGrid.EmergencyStop OR Crane.SoftwareEmergency OR Stamp.SoftwareEmergency OR PicAlpha.SoftwareEmergency;
        StartButton := Stack.StartButton OR LargeSortingConveyor.StartButton OR Stamp.StartButton OR SafetyDoor.StartButton OR LightGrid.StartButton;
        Crane.ACT_AutomaticExecute();
        Stack.ACT_AutomaticExecute();
        Stamp.ACT_AutomaticExecute();
        LargeSortingConveyor.ACT_AutomaticExecute();
        PicAlphaConveyor.ACT_AutomaticExecute();
        SmallSortingConveyor.ACT_AutomaticExecute();
        RefillConveyor.ACT_AutomaticExecute();
        PicAlpha.ACT_AutomaticExecute();
    END_ACTION
    ACTION EmergencyStop_entry

        EmergencyHandled:=FALSE;

        LargeSortingConveyor.Panel.ACT_TurnLampWhite_Off();
        Stack.Panel.ACT_TurnLampWhite_Off();
        Stamp.Panel.ACT_TurnLampWhite_Off();
        LargeSortingConveyor.Panel.ACT_TurnLampGreen_Off();
        Stack.Panel.ACT_TurnLampGreen_Off();
        Stamp.Panel.ACT_TurnLampGreen_Off();
    END_ACTION
    ACTION Init_entry

        InitCompleted:=FALSE;

        LargeSortingConveyor.Panel.ACT_TurnLampWhite_On();
        Stack.Panel.ACT_TurnLampWhite_On();
        Stamp.Panel.ACT_TurnLampWhite_On();
        LargeSortingConveyor.Panel.ACT_TurnLampGreen_Off();
        Stack.Panel.ACT_TurnLampGreen_Off();
        Stamp.Panel.ACT_TurnLampGreen_Off();
    END_ACTION
    ACTION Ready_To_Initialise_active

        EmergencyStop := Stack.EmergencyStop OR LargeSortingConveyor.EmergencyStop OR Stamp.EmergencyStop OR SafetyDoor.EmergencyStop OR LightGrid.EmergencyStop OR Crane.SoftwareEmergency OR Stamp.SoftwareEmergency OR PicAlpha.SoftwareEmergency;
        StartButton := Stack.StartButton OR LargeSortingConveyor.StartButton OR Stamp.StartButton OR SafetyDoor.StartButton OR LightGrid.StartButton;
        IF(StartButton)THEN
        	Stamp.SoftwareEmergency:=FALSE;
        	Crane.SoftwareEmergency:=FALSE;
        	PicAlpha.SoftwareEmergency:=FALSE;
        END_IF
    END_ACTION
    ACTION SFC_Reset_active

        (*PPU*)
        	//Variables
        	InitCompleted:=FALSE;
        	AutomaticExecuteCompleted:=FALSE;

        (*Crane Reset*)
        	Crane(SFCReset:=TRUE);
        	Crane.ACT_Init(SFCReset:=TRUE);
        	Crane.ACT_AutomaticExecute(SFCReset:=TRUE);
        	Crane.ACT_EmergencyStop(SFCReset:=TRUE);
        	Crane.ACT_MoveToConveyor(SFCReset:=TRUE);
        	Crane.ACT_MoveToStack(SFCReset:=TRUE);
        	Crane.ACT_MoveToStamp(SFCReset:=TRUE);
        	Crane.ACT_PickUpWP(SFCReset:=TRUE);
        	Crane.ACT_PutDownWP(SFCReset:=TRUE);

        (*LargeSortingConveyor Reset*)
        	LargeSortingConveyor(SFCReset:=TRUE);
        	LargeSortingConveyor.ACT_Init(SFCReset:=TRUE);
        	LargeSortingConveyor.ACT_AutomaticExecute(SFCReset:=TRUE);
        	LargeSortingConveyor.ACT_ChangeTarget(SFCReset:=TRUE);
        	LargeSortingConveyor.ACT_CheckWPType(SFCReset:=TRUE);
        	LargeSortingConveyor.ACT_SortWP(SFCReset:=TRUE);

        (*Stack Reset*)
        	Stack(SFCReset:=TRUE);
        	Stack.ACT_Init(SFCReset:=TRUE);
        	Stack.ACT_AutomaticExecute(SFCReset:=TRUE);
        	Stack.ACT_ProvideWP(SFCReset:=TRUE);

        (*Stamp Reset*)
        	Stamp(SFCReset:=TRUE);
        	Stamp.ACT_Init(SFCReset:=TRUE);
        	Stamp.ACT_AutomaticExecute(SFCReset:=TRUE);
        	Stamp.ACT_Stamp(SFCReset:=TRUE);

        (*PicAlphaConveyor Reset*)
        	PicAlphaConveyor(SFCReset:=TRUE);
        	PicAlphaConveyor.ACT_Init(SFCReset:=TRUE);
        	PicAlphaConveyor.ACT_AutomaticExecute(SFCReset:=TRUE);
        	PicAlphaConveyor.ACT_SeperateWP(SFCReset:=TRUE);

        (*SmallSortingConveyor Reset*)
        	SmallSortingConveyor(SFCReset:=TRUE);
        	SmallSortingConveyor.ACT_Init(SFCReset:=TRUE);
        	SmallSortingConveyor.ACT_AutomaticExecute(SFCReset:=TRUE);
        	SmallSortingConveyor.ACT_SortWP(SFCReset:=TRUE);
        	SmallSortingConveyor.ACT_ChangeTarget(SFCReset:=TRUE);
        	SmallSortingConveyor.ACT_CheckWPType(SFCReset:=TRUE);

        (*RefillConveyor Reset*)
        	RefillConveyor(SFCReset:=TRUE);
        	RefillConveyor.ACT_Init(SFCReset:=TRUE);
        	RefillConveyor.ACT_AutomaticExecute(SFCReset:=TRUE);
        	RefillConveyor.ACT_SeperateWP(SFCReset:=TRUE);

        (*PicAlpha Reset*)
        	PicAlpha(SFCReset:=TRUE);
        	PicAlpha.ACT_Init(SFCReset:=TRUE);
        	PicAlpha.ACT_AutomaticExecute(SFCReset:=TRUE);
        	PicAlpha.ACT_MoveToPos1(SFCReset:=TRUE);
        	PicAlpha.ACT_MoveToPos2(SFCReset:=TRUE);
        	PicAlpha.ACT_MoveToPos3(SFCReset:=TRUE);
        	PicAlpha.ACT_MoveToPos4(SFCReset:=TRUE);
        	PicAlpha.ACT_PickUpWP(SFCReset:=TRUE);
        	PicAlpha.ACT_PutDownWP(SFCReset:=TRUE);

        SFCResetCompleted:=TRUE;
    END_ACTION
    ACTION SFC_Reset_entry

        SFCResetCompleted:=FALSE;
        GVL.IsSFCResetting:=TRUE;
    END_ACTION
    ACTION SFC_Reset_Reset_active

        (*Crane Reset*)
        	Crane(SFCReset:=FALSE);
        	Crane.ACT_Init(SFCReset:=FALSE);
        	Crane.ACT_AutomaticExecute(SFCReset:=FALSE);
        	Crane.ACT_EmergencyStop(SFCReset:=FALSE);
        	Crane.ACT_MoveToConveyor(SFCReset:=FALSE);
        	Crane.ACT_MoveToStack(SFCReset:=FALSE);
        	Crane.ACT_MoveToStamp(SFCReset:=FALSE);
        	Crane.ACT_PickUpWP(SFCReset:=FALSE);
        	Crane.ACT_PutDownWP(SFCReset:=FALSE);
        	Crane.LiftingCylinder.ACT_Retract();
        	Crane.Gripper.ACT_Release();
        	Crane.Table.Motor.ACT_Stop();
        	//Variables
        	Crane.SFCReset:=FALSE;

        (*LargeSortingConveyor Reset*)
        	LargeSortingConveyor(SFCReset:=FALSE);
        	LargeSortingConveyor.ACT_Init(SFCReset:=FALSE);
        	LargeSortingConveyor.ACT_AutomaticExecute(SFCReset:=FALSE);
        	LargeSortingConveyor.ACT_ChangeTarget(SFCReset:=FALSE);
        	LargeSortingConveyor.ACT_CheckWPType(SFCReset:=FALSE);
        	LargeSortingConveyor.ACT_SortWP(SFCReset:=FALSE);
        	LargeSortingConveyor.Motor.ACT_Stop();
        	LargeSortingConveyor.Seperator1.ACT_Retract();
        	LargeSortingConveyor.Seperator2.ACT_Retract();
        	//Variables
        	LargeSortingConveyor.SFCReset:=FALSE;

        (*Stack Reset*)
        	Stack(SFCReset:=FALSE);
        	Stack.ACT_Init(SFCReset:=FALSE);
        	Stack.ACT_AutomaticExecute(SFCReset:=FALSE);
        	Stack.ACT_ProvideWP(SFCReset:=FALSE);
        	Stack.Seperator.ACT_Retract();
        	//Variables
        	Stack.SFCReset:=FALSE;

        (*Stamp Reset*)
        	Stamp(SFCReset:=FALSE);
        	Stamp.ACT_Init(SFCReset:=FALSE);
        	Stamp.ACT_AutomaticExecute(SFCReset:=FALSE);
        	Stamp.ACT_Stamp(SFCReset:=FALSE);
        	Stamp.StampingCylinder.ACT_Retract();
        	Stamp.SlidingCylinder.ACT_Extend();
        	//Variables
        	Stamp.SFCReset:=FALSE;

        (*PicAlphaConveyor Reset*)
        	PicAlphaConveyor(SFCReset:=FALSE);
        	PicAlphaConveyor.ACT_Init(SFCReset:=FALSE);
        	PicAlphaConveyor.ACT_AutomaticExecute(SFCReset:=FALSE);
        	PicAlphaConveyor.ACT_SeperateWP(SFCReset:=FALSE);
        	//Variables
        	PicAlphaConveyor.SFCReset:=FALSE;

        (*SmallSortingConveyor Reset*)
        	SmallSortingConveyor(SFCReset:=FALSE);
        	SmallSortingConveyor.ACT_Init(SFCReset:=FALSE);
        	SmallSortingConveyor.ACT_AutomaticExecute(SFCReset:=FALSE);
        	SmallSortingConveyor.ACT_SortWP(SFCReset:=FALSE);
        	SmallSortingConveyor.ACT_ChangeTarget(SFCReset:=FALSE);
        	SmallSortingConveyor.ACT_CheckWPType(SFCReset:=FALSE);
        	//Variables
        	SmallSortingConveyor.SFCReset:=FALSE;

        (*RefillConveyor Reset*)
        	RefillConveyor(SFCReset:=FALSE);
        	RefillConveyor.ACT_Init(SFCReset:=FALSE);
        	RefillConveyor.ACT_AutomaticExecute(SFCReset:=FALSE);
        	RefillConveyor.ACT_SeperateWP(SFCReset:=FALSE);
        	//Variables
        	RefillConveyor.SFCReset:=FALSE;

        (*PicAlpha Reset*)
        	PicAlpha(SFCReset:=FALSE);
        	PicAlpha.ACT_Init(SFCReset:=FALSE);
        	PicAlpha.ACT_AutomaticExecute(SFCReset:=FALSE);
        	PicAlpha.ACT_MoveToPos1(SFCReset:=FALSE);
        	PicAlpha.ACT_MoveToPos2(SFCReset:=FALSE);
        	PicAlpha.ACT_MoveToPos3(SFCReset:=FALSE);
        	PicAlpha.ACT_MoveToPos4(SFCReset:=FALSE);
        	PicAlpha.ACT_PickUpWP(SFCReset:=FALSE);
        	PicAlpha.ACT_PutDownWP(SFCReset:=FALSE);
        	//Variables
        	PicAlpha.SFCReset:=FALSE;

        SFCResetResetCompleted:=TRUE;
        SFCResetCompleted:=TRUE;
    END_ACTION
    ACTION SFC_Reset_Reset_entry

        SFCResetResetCompleted:=FALSE;
        GVL.IsSFCResetting:=TRUE;
    END_ACTION
    ACTION SFC_Reset_Reset_exit

        GVL.IsSFCResetting:=FALSE;
    END_ACTION
    ACTION ACT_AutomaticExecute

        INITIAL_STEP AutomaticExecute_Init : (*Local Id: 0 *)
        END_STEP

        STEP Call_All : (*Local Id: 3 *)
            CallAll_AutomationExecutes(N);
        END_STEP
        TRANSITION FROM (AutomaticExecute_Init) TO (Call_All) := (Not AutomaticExecuteCompleted AND SFCResetCompleted AND NOT GVL.IsSFCResetting); END_TRANSITION
        TRANSITION FROM (Call_All) TO (AutomaticExecute_Init) := (AutomaticExecuteCompleted); END_TRANSITION
    END_ACTION
    ACTION ACT_EmergencyStop

        INITIAL_STEP EmergencyStop_Init : (*Local Id: 0 *)
        END_STEP

        STEP Stack_ES : (*Local Id: 3 *)
            Stack.ACT_EmergencyStop(N);
        END_STEP

        STEP Crane_ES : (*Local Id: 6 *)
            Crane.ACT_EmergencyStop(N);
        END_STEP

        STEP LargeSortingConveyor_ES : (*Local Id: 9 *)
            LargeSortingConveyor.ACT_EmergencyStop(N);
        END_STEP

        STEP PicAlphaConveyor_ES : (*Local Id: 12 *)
            PicAlphaConveyor.ACT_EmergencyStop(N);
        END_STEP

        STEP SmallSortingConveyor_ES : (*Local Id: 15 *)
            SmallSortingConveyor.ACT_EmergencyStop(N);
        END_STEP

        STEP RefillConveyor_ES : (*Local Id: 18 *)
            RefillConveyor.ACT_EmergencyStop(N);
        END_STEP

        STEP Stamp_ES : (*Local Id: 21 *)
            Stamp.ACT_EmergencyStop(N);
        END_STEP

        STEP PicAlpha_ES : (*Local Id: 24 *)
            PicAlpha.ACT_EmergencyStop(N);
        END_STEP

        STEP Emergency_Handled : (*Local Id: 27 *)
        END_STEP
        TRANSITION FROM (EmergencyStop_Init) TO (Stack_ES) := (NOT EmergencyHandled AND NOT GVL.IsSFCResetting); END_TRANSITION
        TRANSITION FROM (Stack_ES) TO (Crane_ES) := (Stack.EmergencyHandled); END_TRANSITION
        TRANSITION FROM (Crane_ES) TO (LargeSortingConveyor_ES) := (Crane.EmergencyHandled); END_TRANSITION
        TRANSITION FROM (LargeSortingConveyor_ES) TO (PicAlphaConveyor_ES) := (LargeSortingConveyor.EmergencyHandled); END_TRANSITION
        TRANSITION FROM (PicAlphaConveyor_ES) TO (SmallSortingConveyor_ES) := (PicAlphaConveyor.EmergencyHandled); END_TRANSITION
        TRANSITION FROM (SmallSortingConveyor_ES) TO (RefillConveyor_ES) := (SmallSortingConveyor.EmergencyHandled); END_TRANSITION
        TRANSITION FROM (RefillConveyor_ES) TO (Stamp_ES) := (RefillConveyor.EmergencyHandled); END_TRANSITION
        TRANSITION FROM (Stamp_ES) TO (PicAlpha_ES) := (Stamp.EmergencyHandled); END_TRANSITION
        TRANSITION FROM (PicAlpha_ES) TO (Emergency_Handled) := (PicAlpha.EmergencyHandled); END_TRANSITION
        TRANSITION FROM (Emergency_Handled) TO (EmergencyStop_Init) := (EmergencyHandled); END_TRANSITION
    END_ACTION
    ACTION ACT_Init

        INITIAL_STEP Initialisation_Init : (*Local Id: 0 *)
        END_STEP

        STEP Stamp_Init : (*Local Id: 6 *)
            Stamp.ACT_Init(N);
        END_STEP

        STEP Crane_Init : (*Local Id: 9 *)
            Crane.ACT_Init(N);
        END_STEP

        STEP PicAlpha_Init : (*Local Id: 12 *)
            PicAlpha.ACT_Init(N);
        END_STEP

        STEP LargeSortingConveyor_Init : (*Local Id: 16 *)
            LargeSortingConveyor.ACT_Init(N);
        END_STEP

        STEP PicAlphaConveyor_Init : (*Local Id: 17 *)
            PicAlphaConveyor.ACT_Init(N);
        END_STEP

        STEP SmallSortingConveyor_Init : (*Local Id: 18 *)
            SmallSortingConveyor.ACT_Init(N);
        END_STEP

        STEP RefillConveoyr_Init : (*Local Id: 19 *)
            RefillConveyor.ACT_Init(N);
        END_STEP

        STEP Stack_Init : (*Local Id: 23 *)
            Stack.ACT_Init(N);
        END_STEP

        STEP Init_Completed : (*Local Id: 26 *)
        END_STEP

        STEP EmergencyChecking : (*Local Id: 29 *)
            ACT_CheckEmergency(N);
        END_STEP
        TRANSITION FROM (Initialisation_Init) TO (Stamp_Init, EmergencyChecking) := (NOT InitCompleted AND NOT GVL.IsSFCResetting); END_TRANSITION
        TRANSITION FROM (PicAlpha_Init) TO (LargeSortingConveyor_Init, PicAlphaConveyor_Init, SmallSortingConveyor_Init, RefillConveoyr_Init) := (PicAlpha.InitCompleted); END_TRANSITION
        TRANSITION FROM (LargeSortingConveyor_Init, PicAlphaConveyor_Init, SmallSortingConveyor_Init, RefillConveoyr_Init) TO (Stack_Init) := (LargeSortingConveyor.InitCompleted); END_TRANSITION
        TRANSITION FROM (Init_Completed, EmergencyChecking) TO (Initialisation_Init) := (InitCompleted); END_TRANSITION
        TRANSITION FROM (Stamp_Init) TO (Crane_Init) := (Stamp.InitCompleted); END_TRANSITION
        TRANSITION FROM (Crane_Init) TO (PicAlpha_Init) := (Crane.InitCompleted); END_TRANSITION
        TRANSITION FROM (Stack_Init) TO (Init_Completed) := (Stack.InitCompleted); END_TRANSITION
    END_ACTION

    INITIAL_STEP Init : (*Local Id: 0 *)
    END_STEP

    STEP SFC_Reset_Reset : (*Local Id: 3 *)
        SFC_Reset_Reset_entry(P0);
        SFC_Reset_Reset_exit(P1);
        SFC_Reset_Reset_active(N);
    END_STEP

    STEP Start : (*Local Id: 6 *)
        ACT_Start(N);
    END_STEP

    STEP Initialisation_2 : (*Local Id: 9 *)
        Init_entry(P0);
        ACT_Init(N);
    END_STEP

    STEP AutomaticExecute : (*Local Id: 17 *)
        AutomaticExecute_entry(P0);
        ACT_AutomaticExecute(N);
    END_STEP

    STEP Emergency_Stop : (*Local Id: 25 *)
        EmergencyStop_entry(P0);
        ACT_EmergencyStop(N);
    END_STEP

    STEP SFC_Reset : (*Local Id: 28 *)
        SFC_Reset_entry(P0);
        SFC_Reset_active(N);
    END_STEP

    STEP Ready_To_Initialise : (*Local Id: 31 *)
        Ready_To_Initialise_active(N);
    END_STEP
    TRANSITION FROM (Initialisation_2) TO (AutomaticExecute) := (InitCompleted); END_TRANSITION
    TRANSITION FROM (Initialisation_2) TO (Emergency_Stop) := (EmergencyStop); END_TRANSITION
    TRANSITION FROM (AutomaticExecute) TO (Emergency_Stop) := (EmergencyStop); END_TRANSITION
    TRANSITION FROM (AutomaticExecute) TO (Init) := (StartButton); END_TRANSITION
    TRANSITION FROM (Initialisation_2) TO (AutomaticExecute) := (InitCompleted); END_TRANSITION
    TRANSITION FROM (AutomaticExecute) TO (Emergency_Stop) := (EmergencyStop); END_TRANSITION
    TRANSITION FROM (Init) TO (SFC_Reset_Reset) := (TRUE); END_TRANSITION
    TRANSITION FROM (SFC_Reset_Reset) TO (Start) := (SFCResetResetCompleted); END_TRANSITION
    TRANSITION FROM (Start) TO (Initialisation_2) := (StartButton); END_TRANSITION
    TRANSITION FROM (Emergency_Stop) TO (SFC_Reset) := (EmergencyHandled); END_TRANSITION
    TRANSITION FROM (SFC_Reset) TO (Ready_To_Initialise) := (SFCResetCompleted); END_TRANSITION
    TRANSITION FROM (Ready_To_Initialise) TO (Init) := (NOT EmergencyStop); END_TRANSITION
END_FUNCTION_BLOCK

PROGRAM MAIN

    VAR
        xPPU : xPPU;
        Check_Stack_WPPickedUp : BOOL;
        Stack_WPProvided : BOOL;
        Stack_WPType_Black : BOOL;
        Stack_WPType_White : BOOL;
        Stack_WPType_Metallic : BOOL;
        Stack_WPWeight_Light : BOOL;
        Stack_WPWeight_Medium : BOOL;
        Stack_WPWeight_Heavy : BOOL;
        Check_Stack_WPProvided : BOOL;
        Check_Stack_WPType_Black : BOOL;
        Check_Stack_WPType_White : BOOL;
        Check_Stack_WPType_Metallic : BOOL;
        Check_LargeSortingConveyor_IsSorting : BOOL;
        Check_LargeSortingConveyor_AutomaticExecuteCompleted : BOOL;
        Check_Stamp_IsStamping : BOOL;
        Check_Stamp_WPAvailable : BOOL;
        Check_Stamp_AutomaticExecuteCompleted : BOOL;
        Check_RefillConveyor_IsSending : BOOL;
        Crane_WPType_Black : BOOL;
        Crane_WPType_White : BOOL;
        Crane_WPType_Metallic : BOOL;
        Crane_WPWeight_Light : BOOL;
        Crane_WPWeight_Medium : BOOL;
        Crane_WPWeight_Heavy : BOOL;
        Crane_Conveyor_AllowedToOperate : BOOL;
        Crane_Stamp_AllowedToOperate : BOOL;
        Crane_WPPickedUp : BOOL;
        Check_Stamp_AllowedToOperate : BOOL;
        Check_Stamp_WPWeight_Light : BOOL;
        Check_Stamp_WPWeight_Medium : BOOL;
        Check_Stamp_WPWeight_Heavy : BOOL;
        Stamp_WPType_Black : BOOL;
        Stamp_WPType_White : BOOL;
        Stamp_WPType_Metallic : BOOL;
        Stamp_WPWeight_Light : BOOL;
        Stamp_WPWeight_Medium : BOOL;
        Stamp_WPWeight_Heavy : BOOL;
        Stamp_IsStamping : BOOL;
        Stamp_WPAvailable : BOOL;
        Stamp_AutomaticExecuteCompleted : BOOL;
        Check_LargeSortingConveyor_AllowedToOperate : BOOL;
        Check_LargeSortingConveyor_FollowConveyorInitCompleted : BOOL;
        Check_LargeSortingConveyor_FollowConveyorAutoamticExecuteCompleted : BOOL;
        LargeSortingConveyor_InitCompleted : BOOL;
        LargeSortingConveyor_NumberOfWPsAtConveyor : USINT;
        LargeSortingConveyor_FollowConveyor_AllowedToInit : BOOL;
        LargeSortingConveyor_FollowConveyor_AllowedToOperate : BOOL;
        LargeSortingConveyor_IsSorting : BOOL;
        LargeSortingConveyor_AutomaticExecuteCompleted : BOOL;
        Check_PicAlphaConveyor_AllowedToInit : BOOL;
        Check_PicAlphaConveyor_AllowedToReceive : BOOL;
        Check_PicAlphaConveyor_AllowedToSend : BOOL;
        Check_PicAlphaConveyor_FollowConveyor_InitCompleted : BOOL;
        Check_PicAlphaConveyor_PicAlpha_AutomaticExecuteCompleted : BOOL;
        Check_PicAlphaConveyor_FollowConveyor_AutomaticExecuteCompleted : BOOL;
        PicAlphaConveyor_InitCompleted : BOOL;
        PicAlphaConveyor_FollowConveyor_AllowedToInit : BOOL;
        PicAlphaConveyor_PicAlpha_AllowedToOperate : BOOL;
        PicAlphaConveyor_FollowConveyor_AllowedToOperate : BOOL;
        PicAlphaConveyor_AutomaticExecuteReceivingCompleted : BOOL;
        PicAlphaConveyor_AutomaticExecuteSendingCompleted : BOOL;
        Check_SmallSortingConveyor_AllowedToInit : BOOL;
        Check_SmallSortingConveyor_AllowedToOperate : BOOL;
        Check_SmallSortingConveyor_FollowConveyor_InitCompleted : BOOL;
        Check_SmallSortingConveyor_FollowConveyor_AutomaticExecuteCompleted : BOOL;
        SmallSortingConveyor_InitCompleted : BOOL;
        SmallSortingConveyor_FollowConveyor_AllowedToInit : BOOL;
        SmallSortingConveyor_FollowConveyor_AllowedToOperate : BOOL;
        SmallSortingConveyor_AutomaticExecuteCompleted : BOOL;
        SmallSortingConveyor_IsSorting : BOOL;
        Check_RefillConveyor_AllowedToInit : BOOL;
        Check_RefillConveyor_AllowedToReceive : BOOL;
        Check_RefillConveyor_AllowedToSend : BOOL;
        Check_RefillConveyor_FollowConveyor_InitCompleted : BOOL;
        Check_RefillConveyor_FollowConveyor_AutomaticExecuteCompleted : BOOL;
        RefillConveyor_InitCompleted : BOOL;
        RefillConveyor_FollowConveyor_AllowedToInit : BOOL;
        RefillConveyor_FollowConveyor_AllowedToOperate : BOOL;
        RefillConveyor_AutomaticExecuteReceivingCompleted : BOOL;
        RefillConveyor_IsSending : BOOL;
        RefillConveyor_AutomaticExecuteSendingCompleted : BOOL;
        Check_PicAlpha_AllowedToOperate : BOOL;
        Check_PicAlpha_Conveyor_AutomaticExecuteCompleted : BOOL;
        PicAlpha_InitCompleted : BOOL;
        PicAlpha_Conveyor_AllowedToOperate : BOOL;
        PicAlpha_AutomaticExecuteCompleted : BOOL;
    END_VAR

    xPPU();
    xPPU.Stack();
    xPPU.Crane();
    xPPU.Stamp();
    xPPU.LargeSortingConveyor();
    xPPU.PicAlphaConveyor();
    xPPU.SmallSortingConveyor();
    xPPU.RefillConveyor();
    xPPU.PicAlpha();
    xPPU.SafetyDoor();
    xPPU.LightGrid();

    //Stack
    	//Waiting for Signals
    	Check_Stack_WPPickedUp := xPPU.Crane.Table.AtStack.DI_SwitchTrue AND xPPU.Crane.WPPickedUp;
    	//Giving Signals
    	Stack_WPProvided := xPPU.Stack.WPProvided;
    	Stack_WPType_Black := xPPU.Stack.WPType_Black;
    	Stack_WPType_White := xPPU.Stack.WPType_White;
    	Stack_WPType_Metallic := xPPU.Stack.WPType_Metallic;
    	Stack_WPWeight_Light := xPPU.Stack.WPWeight_Light;
    	Stack_WPWeight_Medium := xPPU.Stack.WPWeight_Medium;
    	Stack_WPWeight_Heavy := xPPU.Stack.WPWeight_Heavy;
    //Crane
    	//Waiting for Signals
    	Check_Stack_WPProvided := Stack_WPProvided;
    	Check_Stack_WPType_Black := Stack_WPType_Black;
    	Check_Stack_WPType_White := Stack_WPType_White;
    	Check_Stack_WPType_Metallic := Stack_WPType_Metallic;
    	Check_LargeSortingConveyor_IsSorting := LargeSortingConveyor_IsSorting;
    	Check_LargeSortingConveyor_AutomaticExecuteCompleted := LargeSortingConveyor_AutomaticExecuteCompleted;
    	Check_Stamp_IsStamping := Stamp_IsStamping;
    	Check_Stamp_WPAvailable := Stamp_WPAvailable;
    	Check_Stamp_AutomaticExecuteCompleted := Stamp_AutomaticExecuteCompleted;
    	Check_RefillConveyor_IsSending := RefillConveyor_IsSending;
    	//Giving Signals
    	Crane_WPType_Black := xPPU.Crane.WPType_Black;
    	Crane_WPType_White := xPPU.Crane.WPType_White;
    	Crane_WPType_Metallic := xPPU.Crane.WPType_Metallic;
    	Crane_WPWeight_Light := xPPU.Crane.WPWeight_Light;
    	Crane_WPWeight_Medium := xPPU.Crane.WPWeight_Medium;
    	Crane_WPWeight_Heavy := xPPU.Crane.WPWeight_Heavy;
    	Crane_Conveyor_AllowedToOperate := xPPU.Crane.Conveyor_AllowedToOperate;
    	Crane_Stamp_AllowedToOperate := xPPU.Crane.Stamp_AllowedToOperate;
    	Crane_WPPickedUp := xPPU.Crane.Gripper.VacuumSwitch.DI_TakenIn;
    //Stamp
    	//Waiting for Signals
    	Check_Stamp_AllowedToOperate := Crane_Stamp_AllowedToOperate;
    	Check_Stamp_WPWeight_Light := Crane_WPWeight_Light;
    	Check_Stamp_WPWeight_Medium := Crane_WPWeight_Medium;
        Check_Stamp_WPWeight_Heavy := Crane_WPWeight_Heavy;
    	//Giving Signals
    	Stamp_WPType_Black := xPPU.Stamp.WPType_Black;
    	Stamp_WPType_White := xPPU.Stamp.WPType_White;
    	Stamp_WPType_Metallic := xPPU.Stamp.WPType_Metallic;
    	Stamp_WPWeight_Light := xPPU.Stamp.WPWeight_Light;
    	Stamp_WPWeight_Medium := xPPU.Stamp.WPWeight_Medium;
    	Stamp_WPWeight_Heavy := xPPU.Stamp.WPWeight_Heavy;
    	Stamp_IsStamping := xPPU.Stamp.IsStamping;
    	Stamp_WPAvailable := xPPU.Stamp.WPAvailable.DI_SwitchTrue;
    	Stamp_AutomaticExecuteCompleted	:= xPPU.Stamp.AutomaticExecuteCompleted;
    //LargeSortingConveyor
    	//Waiting for Signals
    	Check_LargeSortingConveyor_AllowedToOperate := Crane_Conveyor_AllowedToOperate OR RefillConveyor_FollowConveyor_AllowedToOperate;
    	Check_LargeSortingConveyor_FollowConveyorInitCompleted := PicALphaConveyor_InitCompleted;
    	Check_LargeSortingConveyor_FollowConveyorAutoamticExecuteCompleted := PicALphaConveyor_AutomaticExecuteReceivingCompleted;
    	//Giving Signals
    	LargeSortingConveyor_NumberOfWPsAtConveyor := xPPU.LargeSortingConveyor.NumberOfWPsAtConveyor;
    	LargeSortingConveyor_FollowConveyor_AllowedToInit := xPPU.LargeSortingConveyor.FollowConveyor_AllowedToInit;
    	LargeSortingConveyor_FollowConveyor_AllowedToOperate:= xPPU.LargeSortingConveyor.FollowConveyor_AllowedToOperate;
    	LargeSortingConveyor_IsSorting := xPPU.LargeSortingConveyor.IsSorting;
    	LargeSortingConveyor_AutomaticExecuteCompleted := xPPU.LargeSortingConveyor.AutomaticExecuteCompleted;
    //PicALphaConveyor
    	//Waiting for Signals
    	Check_PicAlphaConveyor_AllowedToInit := LargeSortingConveyor_FollowConveyor_AllowedToInit;
    	Check_PicAlphaConveyor_AllowedToReceive := LargeSortingConveyor_FollowConveyor_AllowedToOperate;
    	Check_PicAlphaConveyor_AllowedToSend := LargeSortingConveyor_NumberOfWPsAtConveyor=3;
    	Check_PicAlphaConveyor_FollowConveyor_InitCompleted := SmallSortingConveyor_InitCompleted;
    	Check_PicAlphaConveyor_PicAlpha_AutomaticExecuteCompleted := PicAlpha_AutomaticExecuteCompleted;
    	Check_PicAlphaConveyor_FollowConveyor_AutomaticExecuteCompleted := SmallSortingConveyor_AutomaticExecuteCompleted;
    	//Giving Signals
    	PicAlphaConveyor_InitCompleted := xPPU.PicALphaConveyor.InitCompleted;
    	PicAlphaConveyor_FollowConveyor_AllowedToInit := xPPU.PicALphaConveyor.FollowConveyor_AllowedToInit;
    	PicAlphaConveyor_PicAlpha_AllowedToOperate := xPPU.PicAlphaConveyor.PicAlpha_AllowedToOperate;
    	PicAlphaConveyor_FollowConveyor_AllowedToOperate := xPPU.PicALphaConveyor.FollowConveyor_AllowedToOperate;
    	PicAlphaConveyor_AutomaticExecuteReceivingCompleted := xPPU.PicALphaConveyor.AutomaticExecuteReceivingCompleted;
    	PicAlphaConveyor_AutomaticExecuteSendingCompleted := xPPU.PicALphaConveyor.AutomaticExecuteSendingCompleted;
    //SmallSortingConveyor
    	//Waiting for Signals
    	Check_SmallSortingConveyor_AllowedToInit := PicALphaConveyor_FollowConveyor_AllowedToInit;
    	Check_SmallSortingConveyor_AllowedToOperate := PicALphaConveyor_FollowConveyor_AllowedToOperate;
    	Check_SmallSortingConveyor_FollowConveyor_InitCompleted := RefillConveyor_InitCompleted;
    	Check_SmallSortingConveyor_FollowConveyor_AutomaticExecuteCompleted := RefillConveyor_AutomaticExecuteReceivingCompleted;
    	//Giving Signals
    	SmallSortingConveyor_InitCompleted := xPPU.SmallSortingConveyor.InitCompleted;
    	SmallSortingConveyor_FollowConveyor_AllowedToInit := xPPU.SmallSortingConveyor.FollowConveyor_AllowedToInit;
    	SmallSortingConveyor_FollowConveyor_AllowedToOperate:= xPPU.SmallSortingConveyor.FollowConveyor_AllowedToOperate;
    	SmallSortingConveyor_AutomaticExecuteCompleted := xPPU.SmallSortingConveyor.AutomaticExecuteCompleted;
    	SmallSortingConveyor_IsSorting := xPPU.SmallSortingConveyor.IsSorting;
    //RefillConveyor
    	//Waiting for Signals
    	Check_RefillConveyor_AllowedToInit := SmallSortingConveyor_FollowConveyor_AllowedToInit;
    	Check_RefillConveyor_AllowedToReceive := SmallSortingConveyor_FollowConveyor_AllowedToOperate;
    	Check_RefillConveyor_AllowedToSend := NOT Crane_WPPickedUp AND NOT LargeSortingConveyor_IsSorting AND NOT Check_LargeSortingConveyor_AllowedToOperate;
    	Check_RefillConveyor_FollowConveyor_InitCompleted := LargeSortingConveyor_InitCompleted;
    	Check_RefillConveyor_FollowConveyor_AutomaticExecuteCompleted := LargeSortingConveyor_AutomaticExecuteCompleted;
    	//Giving Signals
    	RefillConveyor_InitCompleted := xPPU.RefillConveyor.InitCompleted;
    	RefillConveyor_FollowConveyor_AllowedToInit := xPPU.RefillConveyor.FollowConveyor_AllowedToInit;
    	RefillConveyor_FollowConveyor_AllowedToOperate := xPPU.RefillConveyor.FollowConveyor_AllowedToOperate;
    	RefillConveyor_AutomaticExecuteReceivingCompleted := xPPU.RefillConveyor.AutomaticExecuteReceivingCompleted;
    	RefillConveyor_IsSending := xPPU.RefillConveyor.IsSending;
    	RefillConveyor_AutomaticExecuteSendingCompleted := xPPU.RefillConveyor.AutomaticExecuteSendingCompleted;
    //PicAlpha
    	//Waiting for Signals
    	Check_PicAlpha_AllowedToOperate := PicAlphaConveyor_PicAlpha_AllowedToOperate;
    	Check_PicAlpha_Conveyor_AutomaticExecuteCompleted := PicAlphaConveyor_AutomaticExecuteSendingCompleted;
    	//Giving Signals
    	PicAlpha_InitCompleted := xPPU.PicAlpha.InitCompleted;
    	PicAlpha_Conveyor_AllowedToOperate := xPPU.PicAlpha.Conveyor_AllowedToOperate;
    	PicAlpha_AutomaticExecuteCompleted := xPPU.PicAlpha.AutomaticExecuteCompleted;
END_PROGRAM
